Omron CX-Programmer project NewProject (CX-Programmer 9.70)

# PLC NewPLC1: CP1E E20

## Global symbols (name address type ; comment)
0.00 BOOL  ; start
100.00 BOOL  ; output
100.01 BOOL  ; led 2

## Program NewProgram1 (cyclic task 0)

### Section Section1

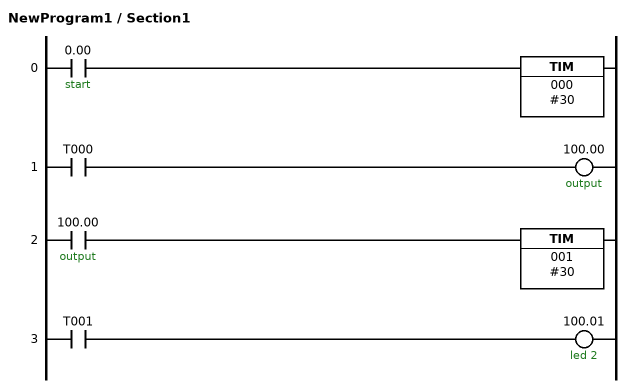
; rung 0
LD 0.00  ; start
TIM 000 #30
; rung 1
LD T000
OUT 100.00  ; output
; rung 2
LD 100.00  ; output
TIM 001 #30
; rung 3
LD T001
OUT 100.01  ; led 2

### Section END
; rung 0
END(001)